	tonFanStart															: TON;
	tonFanRunError														: TON;
	tonInletDoorsOpenError												: TON;
	tonInletDoorsCloseError												: TON;
	tonOutletDoorsOpenError												: TON;
	tonOutletDoorsCloseError											: TON;
	tonInletClampsExtendError											: TON;
	tonInletClampsRetractError											: TON;
	tonOutletClampsExtendError											: TON;
	tonOutletClampsRetractError											: TON;
	tonInletDoorCloseReset												: TON;
	tonOutletDoorCloseReset												: TON;
	
	rRpm																: REAL;
	rRpmOld																: REAL		:= 0;
	rTempTotal															: REAL;
	rTempSP																: REAL;
	rMin																: REAL;
	rMax																: REAL;
	
	byteReactor															: BYTE;
	
	i																	: INT;
	iInletAirSetpoint													: INT		:= 0;
	iTempCount															: INT;
	iHighTempCount														: INT;
	iInletCloseCount													: INT;
	iOutletCloseCount													: INT;
	iInletCount															: ARRAY [0..3] OF INT;
	iOutletCount														: ARRAY [0..3] OF INT;

	bFanRunError														: BOOL;
	bCloseInletDoorsReset												: BOOL;
	bCloseOutletDoorsReset												: BOOL;
	bOpenInletDoors														: BOOL;
	bOpenOutletDoors													: BOOL;
	
    /// <summary>xx01-TT01</summary>
	{attribute 'OPC.UA.DA' := '1'}  				                
	{attribute 'OPC.UA.DA.Access' := '1'}  				                
	inlet_top_left_temp													: REAL;						
    /// <summary>xx01-TT01</summary>
	inlet_top_left_temp_error 											: BOOL;
    /// <summary>inlet top left temp</summary>
	xx01_TT01													AT %I*	: INT;
    /// <summary>inlet top left temp</summary>
	{attribute 'OPC.UA.DA' := '1'}  				                
	{attribute 'OPC.UA.DA.Access' := '1'}  				                
	xx01_TT01_error												AT %I*	: BOOL;
    /// <summary>xx01-TT01</summary>
	{attribute 'OPC.UA.DA' := '1'}  				                
	inlet_top_left_temp_error_or										: BOOL;

    /// <summary>xx01-TT02</summary>
	{attribute 'OPC.UA.DA' := '1'}  				                
	{attribute 'OPC.UA.DA.Access' := '1'}  				                
	inlet_top_right_temp												: REAL;
    /// <summary>xx01-TT02</summary>
	inlet_top_right_temp_error 											: BOOL;
    /// <summary>inlet top right temp</summary>
	xx01_TT02													AT %I*	: INT;
    /// <summary>inlet top right temp</summary>
	{attribute 'OPC.UA.DA' := '1'}  				            	
	{attribute 'OPC.UA.DA.Access' := '1'}  				        	  
	xx01_TT02_error												AT %I*	: BOOL;
    /// <summary>xx01-TT02</summary>
	{attribute 'OPC.UA.DA' := '1'}  				            	
	inlet_top_right_temp_error_or										: BOOL;

    /// <summary>xx01-TT03</summary>
	{attribute 'OPC.UA.DA' := '1'}  				                
	{attribute 'OPC.UA.DA.Access' := '1'}  				                
	inlet_bottom_left_temp												: REAL;						
    /// <summary>xx01-TT03</summary>
	inlet_bottom_left_temp_error 										: BOOL;
    /// <summary>inlet bottom left temp</summary>
	xx01_TT03													AT %I*	: INT;
    /// <summary>inlet bottom left temp</summary>
	{attribute 'OPC.UA.DA' := '1'}  				            	
	{attribute 'OPC.UA.DA.Access' := '1'}  				        	  
	xx01_TT03_error												AT %I*	: BOOL;
    /// <summary>xx01-TT03</summary>
	{attribute 'OPC.UA.DA' := '1'}  				            	
	inlet_bottom_left_temp_error_or										: BOOL;
	
    /// <summary>xx01-TT04</summary>
	{attribute 'OPC.UA.DA' := '1'}  				                
	{attribute 'OPC.UA.DA.Access' := '1'}  				                
	inlet_bottom_right_temp												: REAL;						
    /// <summary>xx01-TT04</summary>
	inlet_bottom_right_temp_error										: BOOL;
    /// <summary>inlet bottom right temp</summary>
	xx01_TT04													AT %I*	: INT;
    /// <summary>inlet bottom right temp</summary>
	{attribute 'OPC.UA.DA' := '1'}  				            	
	{attribute 'OPC.UA.DA.Access' := '1'}  				        	  
	xx01_TT04_error												AT %I*	: BOOL;
    /// <summary>xx01-TT04</summary>
	{attribute 'OPC.UA.DA' := '1'}  				            	
	inlet_bottom_right_temp_error_or									: BOOL;

    /// <summary>xx03-TT01</summary>
	{attribute 'OPC.UA.DA' := '1'}  				                
	{attribute 'OPC.UA.DA.Access' := '1'}  				                
	outlet_top_left_temp												: REAL;						
    /// <summary>xx03-TT01</summary>
	outlet_top_left_temp_error 											: BOOL;
    /// <summary>outlet top left temp</summary>
	xx03_TT01													AT %I*	: INT;
    /// <summary>outlet top left temp</summary>
	{attribute 'OPC.UA.DA' := '1'}  				            	
	{attribute 'OPC.UA.DA.Access' := '1'}  				        	  
	xx03_TT01_error												AT %I*	: BOOL;
    /// <summary>xx03-TT01</summary>
	{attribute 'OPC.UA.DA' := '1'}  				            	
	outlet_top_left_temp_error_or										: BOOL;
	
    /// <summary>xx03-TT02</summary>
	{attribute 'OPC.UA.DA' := '1'}  				                
	{attribute 'OPC.UA.DA.Access' := '1'}  				                
	outlet_top_right_temp												: REAL;
    /// <summary>xx03-TT02</summary>
	outlet_top_right_temp_error 										: BOOL;
    /// <summary>outlet top right temp</summary>
	xx03_TT02													AT %I*	: INT;
    /// <summary>outlet top right temp</summary>
	{attribute 'OPC.UA.DA' := '1'}  				            	
	{attribute 'OPC.UA.DA.Access' := '1'}  				        	  
	xx03_TT02_error												AT %I*	: BOOL;
    /// <summary>xx03-TT02</summary>
	{attribute 'OPC.UA.DA' := '1'}  				            	
	outlet_top_right_temp_error_or										: BOOL;
	
    /// <summary>xx03-TT03</summary>
	{attribute 'OPC.UA.DA' := '1'}  				                
	{attribute 'OPC.UA.DA.Access' := '1'}  				                
	outlet_bottom_left_temp												: REAL;						
    /// <summary>xx03-TT03</summary>
	outlet_bottom_left_temp_error 										: BOOL;
    /// <summary>outlet bottom left temp</summary>
	xx03_TT03													AT %I*	: INT;
    /// <summary>outlet bottom left temp</summary>
	{attribute 'OPC.UA.DA' := '1'}  				            	
	{attribute 'OPC.UA.DA.Access' := '1'}  				        	  
	xx03_TT03_error												AT %I*	: BOOL;
    /// <summary>xx03-TT03</summary>
	{attribute 'OPC.UA.DA' := '1'}  				            	
	outlet_bottom_left_temp_error_or									: BOOL;
	
    /// <summary>xx03-TT04</summary>
	{attribute 'OPC.UA.DA' := '1'}  				                
	{attribute 'OPC.UA.DA.Access' := '1'}  				                
	outlet_bottom_right_temp											: REAL;						
    /// <summary>xx03-TT04</summary>
	outlet_bottom_right_temp_error										: BOOL;
    /// <summary>outlet bottom right temp</summary>
	xx03_TT04													AT %I*	: INT;
    /// <summary>outlet bottom right temp</summary>
	{attribute 'OPC.UA.DA' := '1'}  				            	
	{attribute 'OPC.UA.DA.Access' := '1'}  				        	  
	xx03_TT04_error												AT %I*	: BOOL;
    /// <summary>xx03-TT04</summary>
	{attribute 'OPC.UA.DA' := '1'}  				            	
	outlet_bottom_right_temp_error_or									: BOOL;

    /// <summary>xx02-XV01-SV03</summary>
	{attribute 'OPC.UA.DA' := '1'}  				                
	inlet_door_left_actuator_open_solenoid_valve				AT %Q*	: BOOL;
    /// <summary>xx01-XV01-SV03</summary>
	{attribute 'OPC.UA.DA' := '1'}  				                
	inlet_door_right_actuator_open_solenoid_valve				AT %Q*	: BOOL;
    /// <summary>xx02-XV01-SV04</summary>
	{attribute 'OPC.UA.DA' := '1'}  				                
	inlet_door_left_actuator_close_solenoid_valve				AT %Q*	: BOOL;
    /// <summary>xx01-XV01-SV04</summary>
	{attribute 'OPC.UA.DA' := '1'}  				                
	inlet_door_right_actuator_close_solenoid_valve				AT %Q*	: BOOL;
    /// <summary>xx02-XV03-SV03</summary>
	{attribute 'OPC.UA.DA' := '1'}  				                
	outlet_door_left_actuator_open_solenoid_valve				AT %Q*	: BOOL;
    /// <summary>xx01-XV03-SV03</summary>
	{attribute 'OPC.UA.DA' := '1'}  				                
	outlet_door_right_actuator_open_solenoid_valve				AT %Q*	: BOOL;
    /// <summary>xx02-XV03-SV04</summary>
	{attribute 'OPC.UA.DA' := '1'}  				                
	outlet_door_left_actuator_close_solenoid_valve				AT %Q*	: BOOL;
    /// <summary>xx01-XV03-SV04</summary>
	{attribute 'OPC.UA.DA' := '1'}  				                
	outlet_door_right_actuator_close_solenoid_valve				AT %Q*	: BOOL;

    /// <summary>xx02_XV01_SV01</summary>
	{attribute 'OPC.UA.DA' := '1'}  				                
	inlet_door_left_clamps_extend_solenoid_valve				AT %Q*	: BOOL;
    /// <summary>xx01-XV01-SV01</summary>
	{attribute 'OPC.UA.DA' := '1'}  				                
	inlet_door_right_clamps_extend_solenoid_valve				AT %Q*	: BOOL;
    /// <summary>xx02-XV01-SV02</summary>
	{attribute 'OPC.UA.DA' := '1'}  				                
	inlet_door_left_clamps_retract_solenoid_valve				AT %Q*	: BOOL;
    /// <summary>xx01-XV01_SV02</summary>
	{attribute 'OPC.UA.DA' := '1'}  				                
	inlet_door_right_clamps_retract_solenoid_valve				AT %Q*	: BOOL;
    /// <summary>xx02-XV03-SV01</summary>
	{attribute 'OPC.UA.DA' := '1'}  				                
	outlet_door_left_clamps_extend_solenoid_valve				AT %Q*	: BOOL;
    /// <summary>xx01-XV03-SV01</summary>
	{attribute 'OPC.UA.DA' := '1'}  				                
	outlet_door_right_clamps_extend_solenoid_valve				AT %Q*	: BOOL;
    /// <summary>xx02-XV03-SV02</summary>
	{attribute 'OPC.UA.DA' := '1'}  				                
	outlet_door_left_clamps_retract_solenoid_valve				AT %Q*	: BOOL;
    /// <summary>xx01-XV03-SV02</summary>
	{attribute 'OPC.UA.DA' := '1'}  				                
	outlet_door_right_clamps_retract_solenoid_valve				AT %Q*	: BOOL;

    /// <summary>xx02-XV01-ZS01</summary>
	{attribute 'OPC.UA.DA' := '1'}  				                
	{attribute 'OPC.UA.DA.Access' := '1'}  				                
	inlet_door_left_closed_ls									AT %I*	: BOOL;
    /// <summary>xx02-XV01-ZS01</summary>
	{attribute 'OPC.UA.DA' := '1'}  				                
	{attribute 'OPC.UA.DA.Access' := '1'}  				                
	inlet_door_left_closed												: BOOL;
    /// <summary>xx02-XV01-ZS02</summary>
	{attribute 'OPC.UA.DA' := '1'}  				                
	{attribute 'OPC.UA.DA.Access' := '1'}  				                
	inlet_door_left_open_ls										AT %I*	: BOOL;
    /// <summary>xx01-XV01-ZS01</summary>
	{attribute 'OPC.UA.DA' := '1'}  				                
	{attribute 'OPC.UA.DA.Access' := '1'}  				                
	inlet_door_right_closed_ls									AT %I*	: BOOL;
    /// <summary>xx01-XV01-ZS01</summary>
	{attribute 'OPC.UA.DA' := '1'}  				                
	{attribute 'OPC.UA.DA.Access' := '1'}  				                
	inlet_door_right_closed												: BOOL;
    /// <summary>xx01-XV01-ZS02</summary>
	{attribute 'OPC.UA.DA' := '1'}  				                
	{attribute 'OPC.UA.DA.Access' := '1'}  				                
	inlet_door_right_open_ls									AT %I*	: BOOL;

    /// <summary>xx02-XV03-ZS01</summary>
	{attribute 'OPC.UA.DA' := '1'}  				                
	{attribute 'OPC.UA.DA.Access' := '1'}  				                
	outlet_door_left_closed_ls									AT %I*	: BOOL;
    /// <summary>xx02-XV03-ZS01</summary>
	{attribute 'OPC.UA.DA' := '1'}  				                
	{attribute 'OPC.UA.DA.Access' := '1'}  				                
	outlet_door_left_closed												: BOOL;
    /// <summary>xx02-XV03-ZS02</summary>
	{attribute 'OPC.UA.DA' := '1'}  				                
	{attribute 'OPC.UA.DA.Access' := '1'}  				                
	outlet_door_left_open_ls									AT %I*	: BOOL;
    /// <summary>xx01-XV03-ZS01</summary>
	{attribute 'OPC.UA.DA' := '1'}  				                
	{attribute 'OPC.UA.DA.Access' := '1'}  				                
	outlet_door_right_closed_ls									AT %I*	: BOOL;
    /// <summary>xx01-XV03-ZS01</summary>
	{attribute 'OPC.UA.DA' := '1'}  				                
	{attribute 'OPC.UA.DA.Access' := '1'}  				                
	outlet_door_right_closed											: BOOL;
    /// <summary>xx01-XV03-ZS02</summary>
	{attribute 'OPC.UA.DA' := '1'}  				                
	{attribute 'OPC.UA.DA.Access' := '1'}  				                
	outlet_door_right_open_ls									AT %I*	: BOOL;
	
    /// <summary>xx02-XV01-ZS03</summary>
	{attribute 'OPC.UA.DA' := '1'}  				                
	{attribute 'OPC.UA.DA.Access' := '1'}  				                
	inlet_door_left_clamps_extended_ls							AT %I*	: BOOL;
    /// <summary>xx01-XV01-ZS03</summary>
	{attribute 'OPC.UA.DA' := '1'}  				                
	{attribute 'OPC.UA.DA.Access' := '1'}  				                
	inlet_door_right_clamps_extended_ls							AT %I*	: BOOL;
    /// <summary>xx02-XV03-ZS03</summary>
	{attribute 'OPC.UA.DA' := '1'}  				                
	{attribute 'OPC.UA.DA.Access' := '1'}  				                
	outlet_door_left_clamps_extended_ls							AT %I*	: BOOL;
    /// <summary>xx01-XV03-ZS03</summary>
	{attribute 'OPC.UA.DA' := '1'}  				                
	{attribute 'OPC.UA.DA.Access' := '1'}  				                
	outlet_door_right_clamps_extended_ls						AT %I*	: BOOL;
	
    /// <summary>outlet line temp</summary>
	TT06														AT %I*	: INT;
    /// <summary>outlet line temp</summary>
	{attribute 'OPC.UA.DA' := '1'}  				            	
	{attribute 'OPC.UA.DA.Access' := '1'}  				        	  
	TT06_error													AT %I*	: BOOL;
    /// <summary>TT06</summary>
	{attribute 'OPC.UA.DA' := '1'}  				            	
	outlet_line_temp_error_or											: BOOL;

    /// <summary>VFD01</summary>
	{attribute 'OPC.UA.DA' := '1'}  				                
	fan_vfd_enable														: BOOL :=  TRUE;
    /// <summary>VFD01</summary>
	{attribute 'OPC.UA.DA' := '1'}  				                
	fan_vfd_reset														: BOOL;
    /// <summary>VFD01</summary>
	{attribute 'OPC.UA.DA' := '1'}  				                
	{attribute 'OPC.UA.DA.Access' := '1'}  				                
	fan_vfd_enabled														: BOOL;
    /// <summary>VFD01</summary>
	{attribute 'OPC.UA.DA' := '1'}  				                
	{attribute 'OPC.UA.DA.Access' := '1'}  				                
	fan_vfd_output														: REAL;
    /// <summary>VFD01</summary>
	{attribute 'OPC.UA.DA' := '1'}  				                
	{attribute 'OPC.UA.DA.Access' := '1'}  				                
	fan_vfd_current_amps												: REAL;
    /// <summary>VFD01</summary>
	{attribute 'OPC.UA.DA' := '1'}  				                
	{attribute 'OPC.UA.DA.Access' := '1'}  				                
	fan_vfd_output_current												: REAL;
    /// <summary>VFD01</summary>
	fan_vfd_control												AT %Q*	: WORD;
    /// <summary>VFD01</summary>
	fan_vfd_target_vel											AT %Q*	: WORD;
    /// <summary>VFD01</summary>
	fan_vfd_status												AT %I*	: WORD;
    /// <summary>VFD01</summary>
	fan_vfd_velocity											AT %I*	: WORD;
    /// <summary>VFD01</summary>
	fan_vfd_ecat_state											AT %I*  : BOOL;
    /// <summary>VFD01</summary>
	fan_vfd_current												AT %I*	: DINT;
END_VAR

VAR PERSISTENT
    /// <summary>xx01_TT01</summary>
	{attribute 'OPC.UA.DA' := '1'}
	xx01_TT01_offset													: REAL		:= 0;
    /// <summary>xx01_TT02</summary>
	{attribute 'OPC.UA.DA' := '1'}
	xx01_TT02_offset													: REAL		:= 0;
    /// <summary>xx01_TT03</summary>
	{attribute 'OPC.UA.DA' := '1'}
	xx01_TT03_offset													: REAL		:= 0;
    /// <summary>xx01_TT04</summary>
	{attribute 'OPC.UA.DA' := '1'}
	xx01_TT04_offset													: REAL		:= 0;
    /// <summary>xx03_TT01</summary>
	{attribute 'OPC.UA.DA' := '1'}
	xx03_TT01_offset													: REAL		:= 0;
    /// <summary>xx03_TT02</summary>
	{attribute 'OPC.UA.DA' := '1'}
	xx03_TT02_offset													: REAL		:= 0;
    /// <summary>xx03_TT03</summary>
	{attribute 'OPC.UA.DA' := '1'}
	xx03_TT03_offset													: REAL		:= 0;
    /// <summary>xx03_TT04</summary>
	{attribute 'OPC.UA.DA' := '1'}
	xx03_TT04_offset													: REAL		:= 0;
    /// <summary>TT06</summary>
	{attribute 'OPC.UA.DA' := '1'}
	TT06_offset															: REAL		:= 0;
END_VAR

// P1 - FB_Reactor
// Rev 1.0 - November 2, 2024

IF reset THEN
	inlet_clamps_extend_door_open_error									:= FALSE;
	outlet_clamps_extend_door_open_error								:= FALSE;
	IF inlet_clamps_extend_error THEN
		inlet_door_left_clamps_extend_solenoid_valve					:= FALSE;
		inlet_door_right_clamps_extend_solenoid_valve					:= FALSE;
	END_IF
	IF outlet_clamps_extend_error THEN
		outlet_door_left_clamps_extend_solenoid_valve					:= FALSE;
		outlet_door_right_clamps_extend_solenoid_valve					:= FALSE;
	END_IF
	IF inlet_clamps_retract_error THEN
		inlet_door_left_clamps_retract_solenoid_valve					:= FALSE;
		inlet_door_right_clamps_retract_solenoid_valve					:= FALSE;
	END_IF
	IF outlet_clamps_retract_error THEN
		outlet_door_left_clamps_retract_solenoid_valve					:= FALSE;
		outlet_door_right_clamps_retract_solenoid_valve					:= FALSE;
	END_IF
	inlet_doors_close_error												:= FALSE;
	outlet_doors_close_error											:= FALSE;
	inlet_doors_open_error												:= FALSE;
	outlet_doors_open_error												:= FALSE;
	bOpenInletDoors														:= FALSE;
	bOpenOutletDoors													:= FALSE;
END_IF

outlet_line_temp														:= F_Temperature(TT06, TT06_offset);
outlet_line_temp_error													:= TT06_error AND NOT outlet_line_temp_error_or;
error_code																:= F_Error(error_code, outlet_line_temp_error, errOutletLineTemp);

// SORBENT TEMPERATURE HANDLING
rtrigSorbentErrorCheck(CLK:= MAIN.bHalfSecondPulse);
IF rtrigSorbentErrorCheck.Q THEN
	A_Sorbent_Temperatures();
END_IF

// CLAMPS & DOORS
inlet_clamps_extended_status		  									:= inlet_door_left_clamps_extended_ls AND inlet_door_right_clamps_extended_ls;
inlet_clamps_retracted_status		 									:= NOT inlet_door_left_clamps_extended_ls AND NOT inlet_door_right_clamps_extended_ls;
outlet_clamps_extended_status		 									:= outlet_door_left_clamps_extended_ls AND outlet_door_right_clamps_extended_ls;
outlet_clamps_retracted_status											:= NOT outlet_door_left_clamps_extended_ls AND NOT outlet_door_right_clamps_extended_ls;
clamps_extended_status													:= inlet_clamps_extended_status AND outlet_clamps_extended_status;
clamps_retracted_status													:= inlet_clamps_retracted_status AND outlet_clamps_retracted_status;

fbInletDoorLeftClosed(valve:= inlet_door_left_actuator_close_solenoid_valve, limit_switch:= inlet_door_left_closed_ls, door_closed=> inlet_door_left_closed);
fbInletDoorRightClosed(valve:= inlet_door_right_actuator_close_solenoid_valve, limit_switch:= inlet_door_right_closed_ls, door_closed=> inlet_door_right_closed);
fbOutletDoorLeftClosed(valve:= outlet_door_left_actuator_close_solenoid_valve, limit_switch:= outlet_door_left_closed_ls, door_closed=> outlet_door_left_closed);
fbOutletDoorRightClosed(valve:= outlet_door_right_actuator_close_solenoid_valve, limit_switch:= outlet_door_right_closed_ls, door_closed=> outlet_door_right_closed);


inlet_doors_closed_status												:= inlet_door_left_closed AND inlet_door_right_closed;
inlet_doors_open_status													:= inlet_door_left_open_ls AND inlet_door_right_open_ls;
inlet_doors_closed_or_status											:= inlet_doors_closed_or;
outlet_doors_closed_status	  											:= outlet_door_left_closed AND outlet_door_right_closed;
outlet_doors_open_status												:= outlet_door_left_open_ls AND outlet_door_right_open_ls;
outlet_doors_closed_or_status											:= outlet_doors_closed_or;
doors_closed_status														:= inlet_doors_closed_status AND outlet_doors_closed_status;
doors_open_status														:= inlet_doors_open_status AND outlet_doors_open_status;

rtrigExtendInletClamps(CLK:= extend_inlet_clamps);
IF rtrigExtendInletClamps.Q THEN
	inlet_clamps_extend_door_open_error									:= NOT inlet_doors_closed_status AND NOT inlet_doors_closed_or;
END_IF
error_code																:= F_Error(error_code, inlet_clamps_extend_door_open_error, errInletDoorsNotClosedForClamps);

IF extend_inlet_clamps AND (inlet_doors_closed_status OR inlet_doors_closed_or) THEN
	inlet_door_left_clamps_retract_solenoid_valve						:= FALSE;
	inlet_door_right_clamps_retract_solenoid_valve						:= FALSE;
	inlet_door_left_clamps_extend_solenoid_valve						:= TRUE;
	inlet_door_right_clamps_extend_solenoid_valve						:= TRUE;
ELSIF retract_inlet_clamps THEN
	inlet_door_left_clamps_extend_solenoid_valve						:= FALSE;
	inlet_door_right_clamps_extend_solenoid_valve						:= FALSE;
	inlet_door_left_clamps_retract_solenoid_valve						:= TRUE;
	inlet_door_right_clamps_retract_solenoid_valve						:= TRUE;
END_IF
extend_inlet_clamps														:= FALSE;
retract_inlet_clamps													:= FALSE;

rtrigExtendOutletClamps(CLK:= extend_outlet_clamps);
IF rtrigExtendOutletClamps.Q THEN
	outlet_clamps_extend_door_open_error								:= NOT outlet_doors_closed_status AND NOT outlet_doors_closed_or;
END_IF
error_code																:= F_Error(error_code, outlet_clamps_extend_door_open_error, errOutletDoorsNotClosedForClamps);

IF extend_outlet_clamps AND (outlet_doors_closed_status OR outlet_doors_closed_or) THEN
	outlet_door_left_clamps_retract_solenoid_valve						:= FALSE;                                                  
	outlet_door_right_clamps_retract_solenoid_valve						:= FALSE;                                                  
	outlet_door_left_clamps_extend_solenoid_valve						:= TRUE;                                                      
	outlet_door_right_clamps_extend_solenoid_valve						:= TRUE;                                                      
ELSIF retract_outlet_clamps THEN
	outlet_door_left_clamps_extend_solenoid_valve						:= FALSE;
	outlet_door_right_clamps_extend_solenoid_valve						:= FALSE;
	outlet_door_left_clamps_retract_solenoid_valve						:= TRUE;
	outlet_door_right_clamps_retract_solenoid_valve						:= TRUE;
END_IF
extend_outlet_clamps													:= FALSE;
retract_outlet_clamps													:= FALSE;

clamps_extend_door_open_error											:= inlet_clamps_extend_door_open_error OR outlet_clamps_extend_door_open_error;

tonInletClampsExtendError(IN:= inlet_door_left_clamps_extend_solenoid_valve AND inlet_door_right_clamps_extend_solenoid_valve AND NOT inlet_clamps_extended_status, PT:= REAL_TO_TIME(grClampDelay));
tonInletClampsRetractError(IN:= inlet_door_left_clamps_retract_solenoid_valve AND inlet_door_right_clamps_retract_solenoid_valve AND NOT inlet_clamps_retracted_status, PT:= REAL_TO_TIME(grClampDelay));
tonOutletClampsExtendError(IN:= outlet_door_left_clamps_extend_solenoid_valve AND outlet_door_right_clamps_extend_solenoid_valve AND NOT outlet_clamps_extended_status, PT:= REAL_TO_TIME(grClampDelay));
tonOutletClampsRetractError(IN:= outlet_door_left_clamps_retract_solenoid_valve AND outlet_door_right_clamps_retract_solenoid_valve AND NOT outlet_clamps_retracted_status, PT:= REAL_TO_TIME(grClampDelay));

inlet_clamps_extend_error												:= tonInletClampsExtendError.Q;
error_code																:= F_Error(error_code, inlet_clamps_extend_error, errInletClampsExtend);
inlet_clamps_retract_error												:= tonInletClampsRetractError.Q;
error_code																:= F_Error(error_code, inlet_clamps_retract_error, errInletClampsRetract);
outlet_clamps_extend_error												:= tonOutletClampsExtendError.Q;
error_code																:= F_Error(error_code, outlet_clamps_extend_error, errOutletClampsExtend);
outlet_clamps_retract_error												:= tonOutletClampsRetractError.Q;
error_code																:= F_Error(error_code, outlet_clamps_retract_error, errOutletClampsRetract);

clamps_extend_error														:= inlet_clamps_extend_error OR outlet_clamps_extend_error;
clamps_retract_error													:= inlet_clamps_retract_error OR outlet_clamps_retract_error;

inlet_clamps_retracted_or_status										:= inlet_clamps_retracted_or;
IF inlet_clamps_retracted_status OR inlet_clamps_retracted_or THEN
	IF close_inlet_doors THEN
		inlet_door_left_actuator_open_solenoid_valve					:= FALSE;
		inlet_door_right_actuator_open_solenoid_valve					:= FALSE;
		inlet_door_left_actuator_close_solenoid_valve					:= TRUE;
		inlet_door_right_actuator_close_solenoid_valve					:= TRUE;
		bOpenInletDoors													:= FALSE;;
	ELSIF open_inlet_doors THEN
		inlet_door_left_actuator_close_solenoid_valve					:= FALSE;
		inlet_door_right_actuator_close_solenoid_valve					:= FALSE;
		inlet_door_left_actuator_open_solenoid_valve					:= TRUE;
		inlet_door_right_actuator_open_solenoid_valve					:= TRUE;
		bOpenInletDoors													:= TRUE;
	END_IF
END_IF
open_inlet_doors														:= FALSE;
close_inlet_doors														:= FALSE;
error_code																:= F_Error(error_code, NOT inlet_clamps_retracted_status AND NOT inlet_clamps_retracted_or, errInletClampsNotRetractedForDoors);

outlet_clamps_retracted_or_status										:= outlet_clamps_retracted_or;
IF outlet_clamps_retracted_status OR outlet_clamps_retracted_or THEN
	IF close_outlet_doors THEN
		outlet_door_left_actuator_open_solenoid_valve					:= FALSE;
		outlet_door_right_actuator_open_solenoid_valve					:= FALSE;
		outlet_door_left_actuator_close_solenoid_valve					:= TRUE;
		outlet_door_right_actuator_close_solenoid_valve					:= TRUE;
		bOpenOutletDoors												:= FALSE;
	ELSIF open_outlet_doors THEN
		outlet_door_left_actuator_close_solenoid_valve					:= FALSE;
		outlet_door_right_actuator_close_solenoid_valve					:= FALSE;
		outlet_door_left_actuator_open_solenoid_valve					:= TRUE;
		outlet_door_right_actuator_open_solenoid_valve					:= TRUE;
		bOpenOutletDoors												:= TRUE;
	END_IF
END_IF
open_outlet_doors														:= FALSE;
close_outlet_doors														:= FALSE;
error_code																:= F_Error(error_code, NOT outlet_clamps_retracted_status AND NOT outlet_clamps_retracted_or, errOutletClampsNotRetractedForDoors);


tonInletDoorsCloseError(IN:= inlet_door_left_actuator_close_solenoid_valve AND inlet_door_right_actuator_close_solenoid_valve AND NOT inlet_doors_closed_status, PT:= REAL_TO_TIME(grDoorDelay));
IF tonInletDoorsCloseError.Q THEN
	iInletCloseCount													:= iInletCloseCount + 1;
	IF iInletCloseCount >= SP_door_close_retries_before_error THEN
		iInletCloseCount												:= 0;
		bCloseInletDoorsReset											:= FALSE;
		inlet_doors_close_error											:= TRUE;
		inlet_door_left_actuator_close_solenoid_valve					:= FALSE;
		inlet_door_right_actuator_close_solenoid_valve					:= FALSE;
	ELSE
		bCloseInletDoorsReset											:= TRUE;
		open_inlet_doors												:= TRUE;
	END_IF
END_IF
error_code																:= F_Error(error_code, inlet_doors_close_error, errInletDoorsClose);

tonInletDoorCloseReset(IN:= bCloseInletDoorsReset, PT:= REAL_TO_TIME(SP_door_close_reset_duration * _SECONDS));
IF tonInletDoorCloseReset.Q THEN
	bCloseInletDoorsReset												:= FALSE;
	close_inlet_doors													:= TRUE;
END_IF

tonInletDoorsOpenError(IN:= bOpenInletDoors AND NOT inlet_doors_open_status, PT:= REAL_TO_TIME(grDoorDelay));
IF tonInletDoorsOpenError.Q THEN
	inlet_doors_open_error												:= TRUE;
	inlet_door_left_actuator_open_solenoid_valve						:= FALSE;
	inlet_door_right_actuator_open_solenoid_valve						:= FALSE;
END_IF
error_code																:= F_Error(error_code, inlet_doors_open_error, errInletDoorsOpen);

tonOutletDoorsCloseError(IN:= outlet_door_left_actuator_close_solenoid_valve AND outlet_door_right_actuator_close_solenoid_valve AND NOT outlet_doors_closed_status, PT:= REAL_TO_TIME(grDoorDelay));
IF tonOutletDoorsCloseError.Q THEN
	iOutletCloseCount													:= iOutletCloseCount + 1;
	IF iOutletCloseCount >= SP_door_close_retries_before_error THEN
		iOutletCloseCount												:= 0;
		bCloseOutletDoorsReset											:= FALSE;
		outlet_doors_close_error										:= TRUE;
		outlet_door_left_actuator_close_solenoid_valve					:= FALSE;
		outlet_door_right_actuator_close_solenoid_valve					:= FALSE;
	ELSE
		bCloseOutletDoorsReset											:= TRUE;
		open_outlet_doors												:= TRUE;
	END_IF
END_IF
error_code																:= F_Error(error_code, outlet_doors_close_error, errOutletDoorsClose);

tonOutletDoorCloseReset(IN:= bCloseOutletDoorsReset, PT:= REAL_TO_TIME(SP_door_close_reset_duration * _SECONDS));
IF tonOutletDoorCloseReset.Q THEN
	bCloseOutletDoorsReset												:= FALSE;
	close_outlet_doors													:= TRUE;
END_IF

tonOutletDoorsOpenError(IN:= bOpenOutletDoors AND NOT outlet_doors_open_status, PT:= REAL_TO_TIME(grDoorDelay));
IF tonOutletDoorsOpenError.Q THEN
	outlet_doors_open_error												:= TRUE;
	outlet_door_left_actuator_open_solenoid_valve						:= FALSE;
	outlet_door_right_actuator_open_solenoid_valve						:= FALSE;
END_IF
error_code																:= F_Error(error_code, outlet_doors_open_error, errOutletDoorsOpen);

doors_open_error														:= inlet_doors_open_error OR outlet_doors_open_error;
doors_close_error														:= inlet_doors_close_error OR outlet_doors_close_error;

// FAN
tonFanStart(IN:= fan_vfd <> rRpmOld, PT:= INT_TO_TIME((unit - 1) * _FAN_DELAY_TIME));
IF tonFanStart.Q OR fan_vfd = 0 THEN
	rRpmOld																:= fan_vfd;
	rRpm																:= fan_vfd * _FAN_RPM_FACTOR;
END_IF
fbFan(	Enable_Vfd														:= NOT fan_vfd_ecat_state AND fan_vfd_enable,
		Fault_Reset														:= fan_vfd_reset, 
		Rpm																:= rRpm, 
		Minimum_Speed													:= _FAN_SPEED_MIN,
		Maximum_Speed													:= _FAN_SPEED_MAX, 
		StatusWord														:= fan_vfd_status, 
		ControlWord														=> fan_vfd_control, 
		TargetRpm														=> fan_vfd_target_vel, 
		Ready															=> fan_vfd_enabled,
		Error															=> fan_vfd_error);
		
fan_vfd_output															:= WORD_TO_REAL(fan_vfd_velocity) / _FAN_RPM_FACTOR;
fan_running																:= fan_vfd_velocity > _FAN_ON;
fan_vfd_current_amps													:= DINT_TO_REAL(fan_vfd_current) / 100;
fan_vfd_reset															:= FALSE;


tonFanRunError(IN:= rRPM > 0, PT:= _FAN_START_TIME);
fan_run_error															:= tonFanRunError.Q AND NOT fan_running;
error_code																:= F_Error(error_code, fan_vfd_error, errFanVFD);
error_code																:= F_Error(error_code, fan_run_error, errFanRun);

ACTION A_Sorbent_Temperatures:
// P1 - FB_Reator.A_Sorbent_Temperatures
// Rev 1.0 - October 16, 2024

sorbent_low_temp														:= 1000;
sorbent_high_temp														:= -1000;

rTempTotal																:= 0;
iTempCount																:= 0;

inlet_top_left_temp														:= M_Temperature(xx01_TT01, xx01_TT01_offset, xx01_TT01_error, inlet_top_left_temp_error_or, iInletCount[0], inlet_top_left_temp_error, sorbent_low_temp, sorbent_high_temp, rTempTotal, iTempCount);
inlet_top_right_temp													:= M_Temperature(xx01_TT02, xx01_TT02_offset, xx01_TT02_error, inlet_top_right_temp_error_or, iInletCount[1], inlet_top_right_temp_error, sorbent_low_temp, sorbent_high_temp, rTempTotal, iTempCount);
inlet_bottom_left_temp													:= M_Temperature(xx01_TT03, xx01_TT03_offset, xx01_TT03_error, inlet_bottom_left_temp_error_or, iInletCount[2], inlet_bottom_left_temp_error, sorbent_low_temp, sorbent_high_temp, rTempTotal, iTempCount);
inlet_bottom_right_temp													:= M_Temperature(xx01_TT04, xx01_TT04_offset, xx01_TT04_error, inlet_bottom_right_temp_error_or, iInletCount[3], inlet_bottom_right_temp_error, sorbent_low_temp, sorbent_high_temp, rTempTotal, iTempCount);

outlet_top_left_temp													:= M_Temperature(xx03_TT01, xx03_TT01_offset, xx03_TT01_error, outlet_top_left_temp_error_or, iOutletCount[0], outlet_top_left_temp_error, sorbent_low_temp, sorbent_high_temp, rTempTotal, iTempCount);
outlet_top_right_temp													:= M_Temperature(xx03_TT02, xx03_TT02_offset, xx03_TT02_error, outlet_top_right_temp_error_or, iOutletCount[1], outlet_top_right_temp_error, sorbent_low_temp, sorbent_high_temp, rTempTotal, iTempCount);
outlet_bottom_left_temp													:= M_Temperature(xx03_TT03, xx03_TT03_offset, xx03_TT03_error, outlet_bottom_left_temp_error_or, iOutletCount[2], outlet_bottom_left_temp_error, sorbent_low_temp, sorbent_high_temp, rTempTotal, iTempCount);
outlet_bottom_right_temp												:= M_Temperature(xx03_TT04, xx03_TT04_offset, xx03_TT04_error, outlet_bottom_right_temp_error_or, iOutletCount[3], outlet_bottom_right_temp_error, sorbent_low_temp, sorbent_high_temp, rTempTotal, iTempCount);

error_code																:= F_Error(error_code, inlet_top_left_temp_error, errInletTopLeftTemp);
error_code																:= F_Error(error_code, inlet_top_right_temp_error, errInletTopRightTemp);
error_code																:= F_Error(error_code, inlet_bottom_left_temp_error, errInletBottomLeftTemp);
error_code																:= F_Error(error_code, inlet_bottom_right_temp_error, errInletBottomRightTemp);
error_code																:= F_Error(error_code, outlet_top_left_temp_error, errOutletTopLeftTemp);
error_code																:= F_Error(error_code, outlet_top_right_temp_error, errOutletTopRightTemp);
error_code																:= F_Error(error_code, outlet_bottom_left_temp_error, errOutletBottomLeftTemp);
error_code																:= F_Error(error_code, outlet_bottom_right_temp_error, errOutletBottomRightTemp);

sorbent_average_temp													:= SEL(iTempCount > 0, 0, rTempTotal / iTempCount);

FOR i:= 0 TO 3 DO
	iInletCount[i]														:= iInletCount[i] + 1;
	IF iInletCount[i] > _TEMP_VALID_TIME THEN
		iInletCount[i]													:= _TEMP_VALID_TIME;
	END_IF
	iOutletCount[i]														:= iOutletCount[i] + 1;
	IF iOutletCount[i] > _TEMP_VALID_TIME THEN
		iOutletCount[i]													:= _TEMP_VALID_TIME;
	END_IF
END_FOR

iHighTempCount															:= 0;
rMin																	:= SP_minimum_reasonable_sorbent_TC_reading;
rMax																	:= SP_maximum_reasonable_sorbent_TC_reading;
IF iInletAirSetpoint = 0 THEN
	rTempSP																:= SP_vacuum_cooling_target_temperature;
ELSIF iInletAirSetpoint = 1 THEN
	rTempSP																:= SP_maximum_inlet_air_temperature_during_adsorption;
ELSE
	rTempSP																:= SP_maximum_desorption_sorbent_temperature;
END_IF

iHighTempCount															:= M_Temp_Check(xx01_TT01_Error, inlet_top_left_temp, rTempSP, rMin, rMax, iInletCount[0], iHighTempCount);
iHighTempCount															:= M_Temp_Check(xx01_TT02_Error, inlet_top_right_temp, rTempSP, rMin, rMax, iInletCount[1], iHighTempCount);
iHighTempCount															:= M_Temp_Check(xx01_TT03_Error, inlet_bottom_left_temp, rTempSP, rMin, rMax, iInletCount[2], iHighTempCount);
iHighTempCount															:= M_Temp_Check(xx01_TT04_Error, inlet_bottom_right_temp, rTempSP, rMin, rMax, iInletCount[3], iHighTempCount);
iHighTempCount															:= M_Temp_Check(xx03_TT01_Error, outlet_top_left_temp, rTempSP, rMin, rMax, iOutletCount[0], iHighTempCount);
iHighTempCount															:= M_Temp_Check(xx03_TT02_Error, outlet_top_right_temp, rTempSP, rMin, rMax, iOutletCount[1], iHighTempCount);
iHighTempCount															:= M_Temp_Check(xx03_TT03_Error, outlet_bottom_left_temp, rTempSP, rMin, rMax, iOutletCount[2], iHighTempCount);
iHighTempCount															:= M_Temp_Check(xx03_TT04_Error, outlet_bottom_right_temp, rTempSP, rMin, rMax, iOutletCount[3], iHighTempCount);

IF iInletAirSetpoint = 0 THEN
	vacuum_cooling_high_temp_count										:= iHighTempCount;
ELSIF iInletAirSetpoint = 1 THEN
	adsorption_high_temp_count											:= iHighTempCount;
ELSE
	desorption_high_temp_count											:= iHighTempCount;
END_IF
iInletAirSetpoint														:= SEL(iInletAirSetpoint = 2, iInletAirSetpoint + 1, 0);;
END_ACTION

METHOD M_Temp_Check : INT
VAR_INPUT
	Error																: BOOL;
	Temp																: REAL;
	Setpoint															: REAL;
	Minimum																: REAL;
	Maximum																: REAL;
END_VAR
VAR_IN_OUT
	Count																: INT;
	HighTempCount														: INT;
END_VAR
VAR
END_VAR
// FB_Temp_Check
// Rev 1.0 - September 5, 2024

IF Error OR Temp < Minimum OR Temp > Maximum THEN
	Count																:= 0;
ELSIF Temp > Setpoint THEN
	HighTempCount														:= HighTempCount + 1;
END_IF
M_Temp_Check															:= HighTempCount;
END_METHOD

METHOD M_Temperature : REAL
VAR_INPUT
	Temp																: INT;
	Offset																: REAL;
	ErrorIn																: BOOL;
	ErrorOR																: BOOL;
	Count																: INT;
END_VAR
VAR_IN_OUT
	Error																: BOOL;
	Low																	: REAL;
	High																: REAL;
	Total																: REAL;
	Counter																: INT;
END_VAR
// M_Temperature
// Rev 1.0 - October 16, 2024

M_Temperature															:= F_Temperature(Temp, Offset);
Error																	:= (ErrorIn OR Count < _TEMP_VALID_TIME) AND NOT ErrorOR;
IF NOT ErrorIn THEN
	Low																	:= F_LowestReal(M_Temperature, Low);
	High																:= F_HighestReal(M_Temperature, High, 0, 0);
	Total																:= Total + M_Temperature;
	Counter																:= Counter + 1;
END_IF
END_METHOD

END_FUNCTION_BLOCK

// ---- POUs/Function_Blocks/FB_VFD.TcPOU
FUNCTION_BLOCK FB_VFD
VAR_INPUT
	Enable_Vfd															: BOOL;
	Fault_Reset															: BOOL;
	Rpm																	: REAL;
	Minimum_Speed														: REAL		:= 0;
	Maximum_Speed														: REAL		:= 1800;
	StatusWord															: WORD;
END_VAR
VAR_OUTPUT
	ControlWord															: WORD;
	TargetRpm															: WORD;
	Ready																: BOOL;
	Error																: BOOL;
END_VAR
VAR
	rtrigClear															: R_TRIG;
	rtrigReady															: R_TRIG;
	rtrigRun															: R_TRIG;
	tonReady															: TON;
	tonRun																: TON;
	rRpm																: REAL;
	bEnabled															: BOOL;
	
	VFD_OFF																: WORD										:= 0;
	VFD_CLEAR															: WORD										:= 6;
	VFD_READY															: WORD										:= 7;
	VFD_RUN																: WORD										:= 15;
	VFD_FAULTED															: WORD										:= 8;
	VFD_RESET															: WORD										:= 128;
END_VAR

// FB_VFD
// Rev 1.0 - June 22, 2024

rRpm 																	:= Rpm;

bEnabled																:= Enable_Vfd;
IF rRpm = 0 THEN
	bEnabled															:= FALSE;											// Turn output off if rpm is 0
ELSIF rRpm > Maximum_Speed THEN
	rRpm																:= Maximum_Speed;
ELSIF rRpm < Minimum_Speed THEN
	rRpm																:= Minimum_Speed;
END_IF

rtrigClear(CLK:= bEnabled);
IF rtrigClear.Q THEN
	ControlWord															:= VFD_CLEAR;
END_IF

rtrigReady(CLK:= tonReady.Q);
IF rtrigReady.Q THEN
	ControlWord															:= VFD_READY;
END_IF
tonReady(IN:= ControlWord = VFD_CLEAR, PT:= T#100MS);

rtrigRun(CLK:= tonRun.Q);
IF rtrigRun.Q THEN
	ControlWord															:= VFD_RUN;
END_IF
tonRun(IN:= ControlWord = VFD_READY, PT:= T#100MS);

IF NOT bEnabled AND NOT Fault_Reset THEN
	ControlWord															:= VFD_OFF;
	rtrigReady(CLK:= FALSE);
END_IF

IF Error AND Fault_Reset THEN
	ControlWord															:= VFD_RESET;
END_IF

Ready																	:= ControlWord = VFD_READY OR ControlWord = VFD_RUN OR Enable_Vfd;
TargetRpm																:= SEL(Ready, 0, REAL_TO_WORD(rRpm));

Error																	:= (StatusWord AND VFD_FAULTED) > 0;

END_FUNCTION_BLOCK

// ---- POUs/Function_Blocks/FB_Door_Closed.TcPOU
FUNCTION_BLOCK FB_Door_Closed
VAR_INPUT
	valve																: BOOL;
	limit_switch														: BOOL;
END_VAR
VAR_OUTPUT
	door_closed															: BOOL;
END_VAR
VAR
	ton1																: TON;
	rtrig1																: R_TRIG;
END_VAR

// FB_Door_Closed
// Rev 1.0 - November 2, 2024

ton1(IN:= valve AND limit_switch, PT:= _DOOR_LATCH_CLOSE_TIME);
rtrig1(CLK:= ton1.Q);
IF rtrig1.Q THEN
	door_closed															:= TRUE;
ELSIF NOT valve THEN
	door_closed															:= FALSE;
END_IF

END_FUNCTION_BLOCK

// ---- POUs/Functions/F_Temperature.TcPOU
FUNCTION F_Temperature : REAL
VAR_INPUT
	Input																: INT;
	Offset																: REAL;
END_VAR
VAR
END_VAR

// F_Temperature
// Rev 1.0 - December 28, 2023

F_Temperature															:= INT_TO_REAL(Input) / 10.0 + Offset;

END_FUNCTION

// ---- POUs/Functions/F_Error.TcPOU
FUNCTION F_Error : DWORD
VAR_INPUT
	Error_Code															: DWORD;
	Error_On															: BOOL;
	Error																: INT;
END_VAR
VAR
	Error_Bit															: DWORD;
END_VAR

// F_Error - If Error is true, Error_Code is 
// Rev 1.0 - September 24, 2024

Error_Bit																:= LREAL_TO_DWORD(EXPT(2, Error));
F_Error																	:= SEL(Error_On, Error_Code AND NOT Error_Bit, Error_Code OR Error_Bit);

END_FUNCTION

// ---- POUs/Functions/F_LowestReal.TcPOU
FUNCTION F_LowestReal : REAL
VAR_INPUT
	Value1																: REAL;
	Value2																: REAL;
END_VAR
VAR
END_VAR

// F_LowestReal
// Rev 1.0 - March 14, 2024

F_LowestReal															:= SEL(Value1 < Value2, Value2, Value1);

END_FUNCTION

// ---- POUs/Functions/F_HighestReal.TcPOU
FUNCTION F_HighestReal : REAL
VAR_INPUT
	Value1																: REAL;
	Value2																: REAL;
	Value3																: REAL;
	Value4																: REAL;
END_VAR
VAR
	rValue																: REAL;
END_VAR

// F_HighestReal
// Rev 1.0 - April 25, 2024

rValue																		:= SEL(Value1 > Value2, Value2, Value1);
rValue																		:= SEL(rValue > Value3, Value3, rValue);
F_HighestReal																:= SEL(rValue > Value4, Value4, rValue);

END_FUNCTION

// ---- POUs/Function_Blocks/FB_ValveStatus.TcPOU
FUNCTION_BLOCK FB_ValveStatus
VAR_INPUT
	Input																: BOOL;
	Open																: BOOL;
	Closed																: BOOL;
	Delay																: REAL;
END_VAR
VAR_OUTPUT
	Status																: INT;
END_VAR
VAR
	Timer																: TON;
	LastInput															: BOOL;
END_VAR

// FB_ValveStatus
// Rev 1.0 - October 22, 2024

IF Input <> LastInput THEN
	LastInput															:= Input;
	Timer(IN:= FALSE);
END_IF
IF (Input AND NOT Open) OR (NOT Input AND NOT Closed) THEN
	Timer(IN:= TRUE, PT:= REAL_TO_TIME(Delay));
	IF Timer.Q THEN
		Status															:= 2;
	ELSE
		Status															:= 1;
	END_IF
ELSE
	Status																:= 0;
END_IF

END_FUNCTION_BLOCK

// ---- POUs/Function_Blocks/FB_ValveControl.TcPOU
FUNCTION_BLOCK FB_ValveControl
VAR_INPUT
	Setpoint											: REAL;									// Target value
	Control												: REAL;									// Actual value
	Input												: REAL;									// Value to set output in manual mode
	Input_Increment										: REAL;									// Amount to increase valve position during initial manual (slow) opening
	Full_Output_SP										: REAL;									// Percentage at which slow initial speed stops and valve opens fully
	Minimum_Output										: REAL	:= 0;							// Minimum output in auto mode
	LoopTime											: REAL	:= 500;							// PI loop time in msecs
	Kp													: REAL	:= 100;							// Proportional constant
	Ki													: REAL	:= 0.05;						// Integral constant
	IBand												: REAL	:= 3;							// Plus/minus range within setpoint that Integral is active
	Base												: INT	:= 16384;						// Ideal output to hit setpoint
	BaseAdjust											: INT	:= 10;							// Amount to adjust base value if not within IBand range 
	Mode												: INT	:= 0;							// 0 = Off, 1 = Manual, 2 = Modulation, 3 = Autotune (not currently implemented)
	Closed												: BOOL;
	Error												: BOOL;
	Reverse												: BOOL;
END_VAR                                 		
VAR_OUTPUT                              		
	Output												: INT;
	Mode_Out											: INT;
END_VAR                                 		
VAR                                     		
	bNegativeError										: BOOL;
	bLastError											: BOOL;
	bSlow												: BOOL;
	rInput												: REAL;
	rError												: REAL;
	P													: REAL;
	I													: REAL;
	rBase												: INT;
	MinOut												: INT;
	tonTimer											: TON;
	rtrigManualValveOpen								: R_TRIG;
END_VAR

// FB_ValveControl
// Rev 1.0 - October 24, 2024

MinOut													:= REAL_TO_INT(Minimum_Output * _PERCENT_FACTOR);
IF Mode = eOff OR Mode > eAuto THEN
	Output												:= 0;
	I													:= 0;													// Reset Integral error 
	rBase												:= Base;
ELSIF Mode = eManual THEN
	rtrigManualValveOpen(CLK:= Closed AND Input = 100);
	IF rtrigManualValveOpen.Q THEN
		bSlow											:= TRUE;
		rInput											:= 0;
	END_IF
	IF bSlow THEN
		tonTimer(IN:= TRUE, PT:= T#500MS);
		IF tonTimer.Q THEN
			rInput										:= rInput + Input_Increment;
			rInput										:= SEL(rInput > 100, rInput, 100);
			tonTimer(in:= FALSE);
		END_IF
		Output											:= REAL_TO_INT(rInput * _PERCENT_FACTOR);
		IF rInput >= Full_Output_SP THEN
			bSlow										:= FALSE;
		END_IF
	ELSE
		Output											:= REAL_TO_INT(Input * _PERCENT_FACTOR);
		rBase											:= Base;
	END_IF
ELSIF Mode = eAuto THEN																							// Modulation
	IF tonTimer.Q THEN
		tonTimer(IN:= FALSE);	
		rError											:= SEL(Reverse, Setpoint - Control, Control - Setpoint);
		bNegativeError									:= rError > 0;
		IF bNegativeError <> bLastError THEN																	// Zero crossover
			bLastError									:= bNegativeError;
			rBase										:= REAL_TO_INT(rBase + I);
			rBase										:= SEL(rBase < 0, SEL(rBase > 32767, rBase, 32767), 0);
			I											:= 0;
		END_IF
		P												:= rError * Kp;
		I												:= SEL(ABS(rError) < IBand, 0, I + (rError * Ki));
		IF ABS(rError) > IBand THEN
			rBase										:= SEL(bNegativeError, rBase - BaseAdjust, rBase + BaseAdjust);
			rBase										:= SEL(rBase < 0, SEL(rBase > 32767, rBase, 32767), 0);
		END_IF
		Output											:= REAL_TO_INT(rBase + P + I);
		Output											:= SEL(Output < MinOut, Output, MinOut);
	END_IF
	
	tonTimer(IN:= TRUE, PT:= REAL_TO_TIME(LoopTime));
ELSIF Mode = eTune THEN
	;																											// Autotune (TBC)
END_IF

Mode_Out												:= Mode;
Output													:= SEL(Output < 0, SEL(Output > 32767, Output, 32767), 0);

END_FUNCTION_BLOCK

// ---- POUs/Functions/F_AnalogIn.TcPOU
FUNCTION F_AnalogIn : REAL
VAR_INPUT
	Input																: INT;
	Low																	: REAL;
	High																: REAL;
	Minimum																: REAL;
	Offset																: REAL;
END_VAR
VAR
	Value																: REAL;
END_VAR

// F_AnalogIn
// Rev 1.0 - December 28, 2023

Value																	:= ((High - Low) / 32767.0) * INT_TO_REAL(Input) + Low;		// Determine output based on scale
Value																	:= Value + Offset;											// Adjust for any user offset
F_AnalogIn																:= SEL(ABS(Value) > Minimum, 0, Value);						// Value must be above (or below, if negative) minimum or zero is returned

END_FUNCTION

// ---- POUs/Function_Blocks/FB_ReadWrite_Json.TcPOU
FUNCTION_BLOCK FB_ReadWrite_Json
VAR_INPUT
	i_ExecuteRead : BOOL;
	i_ExecuteWrite : BOOL := FALSE;
	i_Json_FilePath : STRING(255);
    i_JsonStructure : STRING;	
END_VAR
VAR_OUTPUT
	o_ConfigReadDone : BOOL;
	o_ReadError		 : BOOL;
END_VAR
VAR
	jsonWriter : BeckhoffJsonReadWriter.JsonParser;
	jsonReader : BeckhoffJsonReadWriter.JsonParser;
	bErrorWrite : BOOL;
	nErrorNoWrite : UDINT;
	bErrorRead : BOOL;
	nErrorNoRead : UDINT;
	fbEdge :FB_EdgeMonitor;
END_VAR

jsonReader( Execute := i_ExecuteRead,
		File := i_Json_FilePath,
		ParseMethod := 'ReadFile', //  Reads from json file and writes to PLC
		Content := i_JsonStructure,
		Port := 851,
		HasError => bErrorRead,
		ErrorId => nErrorNoRead);
		
jsonWriter( Execute := i_ExecuteWrite,
		File := i_Json_FilePath,
		ParseMethod := 'WriteFile', // Reads from PLC and writes to json file
		Content := i_JsonStructure,
		Port := 851,
		HasError => bErrorWrite,
		ErrorId => nErrorNoWrite);	

o_ReadError := 	bErrorRead;	
o_ConfigReadDone := fbEdge.FallingEdge(i_SignalToMonitor := jsonReader.startProcess.BUSY);

END_FUNCTION_BLOCK

// ---- POUs/Function_Blocks/FB_EdgeMonitor.TcPOU
FUNCTION_BLOCK FB_EdgeMonitor
VAR_INPUT
END_VAR
VAR_OUTPUT
END_VAR
VAR
	fTrig : F_TRIG;
	rTrig : R_TRIG;
END_VAR

METHOD FallingEdge : BOOL
VAR_INPUT
	i_SignalToMonitor : BOOL;
END_VAR
fTrig(CLK := i_SignalToMonitor);
IF fTrig.Q THEN
	FallingEdge := TRUE;
ELSE
	FallingEdge := FALSE;
END_IF
END_METHOD

END_FUNCTION_BLOCK

// ---- POUs/Functions/F_IEConvert.TcPOU
FUNCTION F_IEConvert : REAL
VAR_INPUT
	Input																: INT;
	Factor																: REAL;
END_VAR
VAR
END_VAR

// F_IEConvert
// Rev 1.0 - December 28, 2023

F_IEConvert															:= INT_TO_REAL(Input) / Factor;

END_FUNCTION

// ---- POUs/FB_Reactor_Set_Ext_FAT.TcPOU
FUNCTION_BLOCK FB_Reactor_Set_Ext_FAT EXTENDS FB_Reactor_Set
VAR_INPUT
END_VAR
VAR_OUTPUT
END_VAR
VAR
	fb_ReadJsonFAT : FB_ReadWrite_Json;
	sita_bit1 : BOOL;
END_VAR

fb_ReadJsonFAT(
		i_ExecuteRead := sita_bit1,
		i_Json_FilePath := FAT.json_file_path,
		i_JsonStructure := 'FAT.st_steam_desorption');

//Steam_Desorption_FAT();	

SUPER^();

END_FUNCTION_BLOCK

// ---- POUs/Functions/F_Error_Check.TcPOU
FUNCTION F_Error_Check : INT
VAR_INPUT
	ErrorCode															: DWORD;
	Error																: INT;
END_VAR
VAR
END_VAR

// F_Error_Check
// Rev 1.0 - October 9, 2024


F_Error_Check															:= SEL((ErrorCode AND LREAL_TO_DWORD(EXPT(2, Error))) > 0, 0, DWORD_TO_INT(ErrorCode));

END_FUNCTION

// ---- POUs/Functions/F_Error_Range.TcPOU
FUNCTION F_Error_Range : BOOL
VAR_INPUT
	Error_Code															: DWORD;
	First_Error															: INT;
	Last_Error															: INT;
END_VAR
VAR
END_VAR

// F_Error_Range
// Rev 1.0 - September 18, 2024

F_Error_Range															:= Error_Code >= LREAL_TO_DWORD(EXPT(2, First_Error)) AND Error_Code <= LREAL_TO_DWORD(EXPT(2, Last_Error));

END_FUNCTION

// ---- POUs/Function_Blocks/FB_Watchdog.TcPOU
FUNCTION_BLOCK FB_Watchdog
VAR_INPUT
	i_receiving_plc 		: BOOL;  // TRUE if not the initiating  PLC 
	i_auto_reset_enabled	: BOOL;
	i_reset_error 			: BOOL;
	i_timeout	 			: REAL;	
END_VAR
VAR_OUTPUT
	o_error		: BOOL;
END_VAR
VAR
	in_watchdog 		AT %I* : BOOL;  // from remote PLC
	out_watchdog		AT %I* : BOOL;  // to Remote PLC 
	tmrTimeout			: TON;
	error_reset_trig	: R_TRIG;
END_VAR

error_reset_trig(CLK := i_reset_error);

IF i_receiving_plc THEN 
	tmrTimeout(IN:= out_watchdog = NOT in_watchdog,PT := TO_TIME(i_timeout * 1000));
ELSE
	tmrTimeout(IN:= out_watchdog = in_watchdog,PT := TO_TIME(i_timeout * 1000));
END_IF

IF i_auto_reset_enabled THEN 
	o_error := tmrTimeout.Q;
ELSE
	IF tmrTimeout.Q THEN
		o_error := TRUE;
	END_IF
	IF error_reset_trig.Q THEN
		o_error := FALSE;
	END_IF
END_IF

IF i_receiving_plc THEN 
	out_watchdog := NOT in_watchdog;
ELSE
	out_watchdog := in_watchdog;
END_IF

END_FUNCTION_BLOCK
